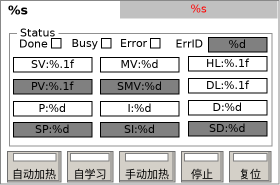
VISUALIZATION HeatModuleVisu  // 280x185
VAR_IN_OUT
	userData:HEATModuleHMI;
END_VAR
    Button (7,151 54x31), "自动加热", input disabled if: NOT userData.HMIEnable
        tap userData.heat
    Rectangle (13,153 43x8), colour toggle: userData.busy
    GroupBox (9,25 263x121), "Status"
        RoundedRectangle (42,13 10x10), colour toggle: userData.done
        RoundedRectangle (92,13 10x10), colour toggle: userData.busy
        RoundedRectangle (141,13 10x10), colour toggle: userData.error
        Rectangle (199,12 59x15), "%d", text variable: userData.errID, input disabled if: true
        Label (164,12 33x14), "ErrID"
        Label (111,12 30x13), "Error"
        Label (62,12 30x13), "Busy"
        Label (9,11 33x16), "Done"
        Rectangle (4,32 79x15), "SV:%.1f", text variable: userData.para_SV
            OnMouseClick: write the text variable via Default, min -10, max 300
        Rectangle (4,54 79x15), "PV:%.1f", text variable: userData.status_PV, input disabled if: true
        Rectangle (91,54 79x15), "SMV:%d", text variable: userData.status_MV, input disabled if: true
        Rectangle (179,53 79x15), "DL:%.1f", text variable: userData.para_LLimit
            OnMouseClick: write the text variable via Default, min -10, max 300
        Rectangle (4,76 79x15), "P:%d", text variable: userData.para_P
            OnMouseClick: write the text variable via Default, min -10, max 300
        Rectangle (91,76 79x15), "I:%d", text variable: userData.para_I
            OnMouseClick: write the text variable via Default, min -10, max 300
        Rectangle (4,97 79x15), "SP:%d", text variable: userData.status_P, input disabled if: true
    Button (67,151 46x31), "自学习", input disabled if: NOT userData.HMIEnable
        tap userData.ATLearning
    Rectangle (70,153 39x8)
    Button (229,151 42x31), "复位"
        tap userData.reset
    Rectangle (233,153 34x8), colour toggle: userData.error
    Rectangle (5,0 112x20), "%s", text variable: userData.nameTXT
    Button (119,151 56x31), "手动加热", input disabled if: false
        tap userData.manuleHeat
    Rectangle (125,153 43x8)
    Button (181,151 42x31), "停止"
        tap userData.stop
    Rectangle (184,153 34x8), colour toggle: userData.stop
    Rectangle (120,0 157x18), "%s", text variable: userData.errTXT
    Rectangle (100,57 79x15), "MV:%d", text variable: userData.para_Manual_MV
        OnMouseClick: write the text variable via Default, min -10, max 300
    Rectangle (188,56 79x15), "HL:%.1f", text variable: userData.para_HLimit
        OnMouseClick: write the text variable via Default, min -10, max 300
    Rectangle (188,100 79x15), "D:%d", text variable: userData.para_D
        OnMouseClick: write the text variable via Default, min -10, max 300
    Rectangle (100,122 79x15), "SI:%d", text variable: userData.status_I, input disabled if: true
    Rectangle (188,121 79x15), "SD:%d", text variable: userData.status_D, input disabled if: true
END_VISUALIZATION

(* stored: Version 1.1.0.1, ProductVersion 3.1.4024.4
   Visu HeatModuleVisu: Id {972414c1-89a1-4faf-a42e-d52e9750453a} *)
